// TIA Portal V17 export
// export: Created 2024-10-03T08:22:49.8034074Z, ExportSetting WithDefaults, DisplayName Totally Integrated Automation Portal, DisplayVersion V17 Update 5, DisplayName TIA Portal Openness, DisplayVersion V17 Update 5, DisplayName TIA Portal Version Control Interface, DisplayVersion V17, DisplayName STEP 7 Professional, DisplayVersion V17 Update 5, DisplayName STEP 7 Safety, DisplayVersion V17, DisplayName WinCC Advanced, DisplayVersion V17 Update 5
VAR_GLOBAL   // PLC tag table "Default tag table"
END_VAR
